FUNCTION_BLOCK FB_Exercice1
VAR_INPUT
END_VAR
VAR_OUTPUT
END_VAR
VAR
	fb_Blinking : ARRAY [0..1] OF FB_Blinking;
END_VAR

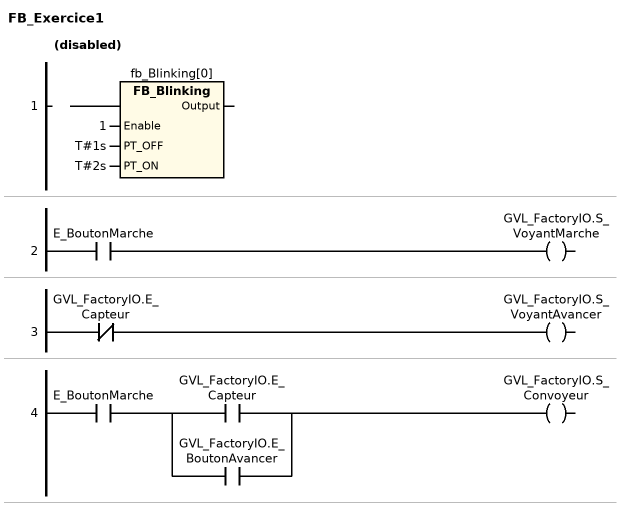
// NETWORK 1 (disabled)
// fb_Blinking[0](Enable := 1, PT_OFF := T#1s, PT_ON := T#2s); // FB_Blinking

// NETWORK 2
GVL_FactoryIO.S_VoyantMarche := E_BoutonMarche;

// NETWORK 3
GVL_FactoryIO.S_VoyantAvancer := NOT GVL_FactoryIO.E_Capteur;

// NETWORK 4
GVL_FactoryIO.S_Convoyeur := E_BoutonMarche AND (GVL_FactoryIO.E_Capteur OR GVL_FactoryIO.E_BoutonAvancer);

END_FUNCTION_BLOCK

(* stored: Version 1.1.0.1, ProductVersion 3.1.4024.11
   POU FB_Exercice1: Id {cc0f096b-f4d5-46dc-ae5e-f73cac9baf65}, SpecialFunc None *)
